// TIA Portal V20 export
DATA_BLOCK "LBP_ConfigData"   // DB7
TITLE = Configuration parameter
{ S7_Optimized_Access := 'FALSE' }
AUTHOR : SINUMERIK
FAMILY : SINUMERIK_ONE
VERSION : 6.14
// Contains parameters for the configuration and initialization of the basic program
// stored: AutoNumber false, InstanceOfName LBP_typeConfigData, InstanceOfType UDT
"LBP_typeConfigData"
   // VAR RETAIN
   //    MCPNum : Int := 1;   // Inputs starting here
   //    MCP1In : Struct   // Pointer
   //       DBNo : Word;
   //       Addr : DWord;
   //    END_STRUCT;
   //    MCP1Out : Struct   // Pointer
   //       DBNo : Word;
   //       Addr : DWord;
   //    END_STRUCT;
   //    reservedByte14_25 : Array[14..25] of Byte;
   //    MCP1BusAdr : Int := 192;
   //    MCP1Timeout : S5Time;
   //    reservedByte30_31 : Array[30..31] of Byte;
   //    MCP2In : Struct   // Pointer
   //       DBNo : Word;
   //       Addr : DWord;
   //    END_STRUCT;
   //    MCP2Out : Struct   // Pointer
   //       DBNo : Word;
   //       Addr : DWord;
   //    END_STRUCT;
   //    reservedByte44_55 : Array[44..55] of Byte;
   //    MCP2BusAdr : Int;
   //    MCP2Timeout : S5Time;
   //    reservedByte60_61 : Array[60..61] of Byte;
   //    reservedBool62_0 : Bool;
   //    MCP1Stop : Bool;
   //    MCP2Stop : Bool;
   //    MCP1NotSend : Bool;
   //    MCP2NotSend : Bool;
   //    reservedBool62_5 : Bool;
   //    reservedBool62_6 : Bool;
   //    MCPBusType : Byte;
   //    HTIf : Int;
   //    HTIn : Struct   // Pointer
   //       DBNo : Word;
   //       Addr : DWord;
   //    END_STRUCT;
   //    HTOut : Struct   // Pointer
   //       DBNo : Word;
   //       Addr : DWord;
   //    END_STRUCT;
   //    reservedByte78_95 : Array[78..95] of Byte;
   //    HTAdr : Int;
   //    reservedByte98_107 : Array[98..107] of Byte;
   //    reservedBool108_0 : Bool;
   //    HTStop : Bool;
   //    HTNotSend : Bool;
   //    NCCyclTimeout : S5Time;
   //    NCRunupTimeout : S5Time;
   //    ListMDecGrp : Int;
   //    reservedBool116_0 : Bool;
   //    MMCToIF : Bool;
   //    HWheelMMC : Bool;
   //    reservedBool116_3 : Bool;
   //    MCP_IF_TCS : Bool;
   //    ExtendChanAxMsg : Bool;
   //    HMIAxisSel : Bool;
   //    DeactivateCtrlEnergy : Bool;
   //    MsgUser : Int := 64;
   //    reservedBool120_0 : Bool;
   //    IRAuxfuT : Bool;
   //    IRAuxfuH : Bool;
   //    IRAuxfuE : Bool;
   //    UserVersion : Struct   // Pointer
   //       DBNo : Word;
   //       Addr : DWord;
   //    END_STRUCT;
   //    OpKeyNum : Int;
   //    Op1KeyIn : Struct   // Pointer
   //       DBNo : Word;
   //       Addr : DWord;
   //    END_STRUCT;
   //    Op1KeyOut : Struct   // Pointer
   //       DBNo : Word;
   //       Addr : DWord;
   //    END_STRUCT;
   //    Op1KeyBusAdr : Int;
   //    Op2KeyIn : Struct   // Pointer
   //       DBNo : Word;
   //       Addr : DWord;
   //    END_STRUCT;
   //    Op2KeyOut : Struct   // Pointer
   //       DBNo : Word;
   //       Addr : DWord;
   //    END_STRUCT;
   //    Op2KeyBusAdr : Int;
   //    Op1KeyStop : Bool;
   //    Op2KeyStop : Bool;
   //    Op1KeyNotSend : Bool;
   //    Op2KeyNotSend : Bool;
   //    reservedByte159 : Byte;
   //    IdentMcpBusAdr : Int;
   //    IdentMcpProfilNo : Byte;
   //    IdentMcpBusType : Byte;
   //    IdentMcpStrobe : Bool;
   //    MaxModeGroup : Int;   // Outputs starting here
   //    MaxChan : Int;
   //    MaxAxis : Int;
   //    ActiveChan : Array[1..10] of Bool;
   //    ActiveAxis : Array[1..31] of Bool;
   //    MaxNumUserDataInt : Int;
   //    MaxNumUserDataHex : Int;
   //    MaxNumUserDataReal : Int;
   //    IdentMcpType : Byte;
   //    IdentMcpLengthIn : Byte;
   //    IdentMcpLengthOut : Byte;
   //    reservedByte188_199 : Array[188..199] of Byte;   // Static starting here
   //    LBPVersionInfo : String[44] := 'SINUMERIK ONE V06.14.00.00.007 13/10/20 $L';
   //    UserVersionInfo : String[44];
   //    GenerateAlarmMsgs : Struct
   //       NumActAlarmMsgs : UInt;
   //       Error : Bool;
   //       StatusID : UInt;
   //       Status : Word;
   //    END_STRUCT;
   //    OpUnitCommId : UInt;   // ID for OpUnitComm
   //    OpUnitInterfaceId : HW_ANY;   // Hardware identifier of Ethernet interface for OpUnitComm
   //    MCP1ConnectionId : CONN_OUC;   // Connection identifier for MCP 1
   //    MCP2ConnectionId : CONN_OUC;   // Connection identifier for MCP 2
   //    HTConnectionId : CONN_OUC;   // Connection identifier for handheld unit
   //    Op1KeyConnectionId : CONN_OUC;   // Connection identifier for Direct Key 1
   //    Op2KeyConnectionId : CONN_OUC;   // Connection identifier for Direct Key 2
   //    IdentConnectionId : CONN_OUC;   // Connection identifier for identification
   //    MCP1LocalUdpPort : UInt;   // Local UDP port for MCP 1
   //    MCP2LocalUdpPort : UInt;   // Local UDP port for MCP 2
   //    HTLocalUdpPort : UInt;   // Local UDP port for handheld unit
   //    Op1KeyLocalUdpPort : UInt;   // Local UDP port for Direct Key 1
   //    Op2KeyLocalUdpPort : UInt;   // Local UDP port for Direct Key 2
   //    IdentLocalUdpPort : UInt;   // Local UDP port for Ident
   //    MCP1Error : Bool;   // Error MCP 1
   //    MCP1Status : Word;   // Error information MCP 1
   //    MCP2Error : Bool;   // Error MCP 2
   //    MCP2Status : Word;   // Error information MCP 2
   //    HTError : Bool;   // Error handheld unit
   //    HTStatus : Word;   // Error information handheld unit
   //    Op1KeyError : Bool;   // Error Direct Key 1
   //    Op1KeyStatus : Word;   // Error information Direct Key 1
   //    Op2KeyError : Bool;   // Error Direct Key 2
   //    Op2KeyStatus : Word;   // Error information Direct Key 2
   //    IdentError : Bool;   // Error identification
   //    IdentStatus : Word;   // Error information Identification
   //    MCP1Ready : Bool;   // MCP1 connected
   //    MCP2Ready : Bool;   // MCP2 connected
   //    HTReady : Bool;   // Handheld unit connected
   //    Op1KeyReady : Bool;   // Direct Key 1 connected
   //    Op2KeyReady : Bool;   // Direct Key 2 connected
   // END_VAR
BEGIN
END_DATA_BLOCK
